Omron CX-Programmer project NewProject (CX-Programmer 9.73)

# PLC NewPLC1: CP1L M

## Global symbols (name address type ; comment)
100.03 BOOL  ; SOAP_APPLICATION
100.04 BOOL  ; BRUSHING
0.05 BOOL  ; SENSOR_5
0.00 BOOL  ; ON_START
0.01 BOOL  ; SENSOR_1
0.02 BOOL  ; SENSOR_2
0.03 BOOL  ; SENSOR_3
0.04 BOOL  ; SENSOR_4
0.06 BOOL  ; STOP_BUTTON
100.00 BOOL  ; INDIKATOR_LAMP
100.01 BOOL  ; KONVEYOR
100.02 BOOL  ; WATER_SPRAYER
100.05 BOOL  ; WATER_WASHER
100.06 BOOL  ; DRYER
T0001 BOOL  ; T1
T0002 BOOL  ; T2
T0003 BOOL  ; T3
T0004 BOOL  ; T4
W100.00 BOOL  ; 0
W100.01 BOOL  ; 1
W100.05 BOOL  ; STOP

## Program NewProgram1 (cyclic task 0)

### Section Section1

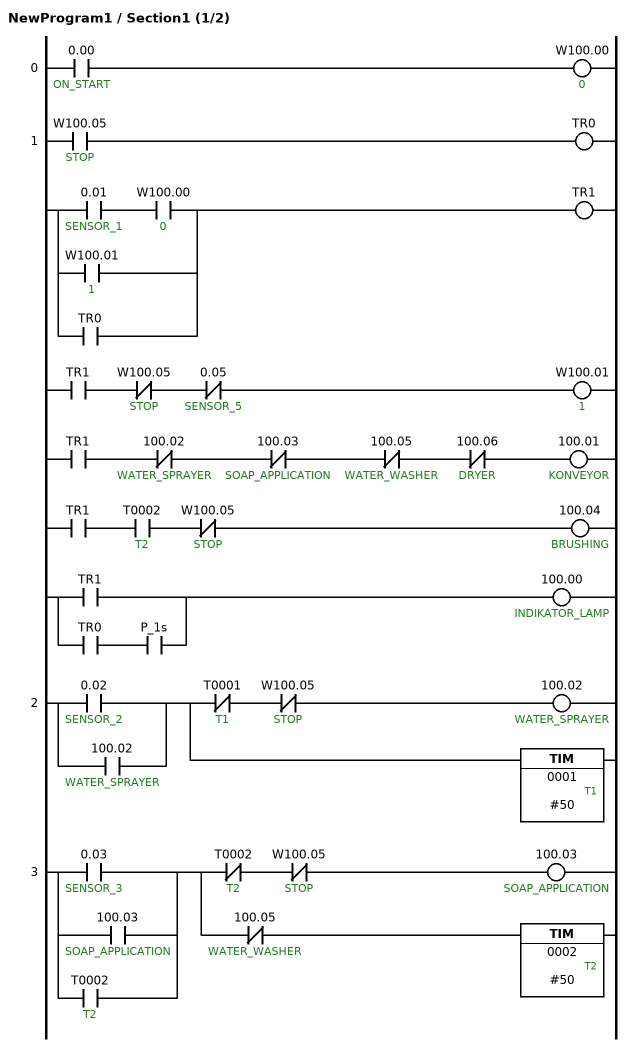
; rung 0
LD 0.00  ; ON_START
OUT W100.00  ; 0
; rung 1
LD 0.01  ; SENSOR_1
AND W100.00  ; 0
OR W100.01  ; 1
LD W100.05  ; STOP
OUT TR0
ORLD
OUT TR1
ANDNOT W100.05  ; STOP
ANDNOT 0.05  ; SENSOR_5
OUT W100.01  ; 1
LD TR1
ANDNOT 100.02  ; WATER_SPRAYER
ANDNOT 100.03  ; SOAP_APPLICATION
ANDNOT 100.05  ; WATER_WASHER
ANDNOT 100.06  ; DRYER
OUT 100.01  ; KONVEYOR
LD TR1
AND T0002  ; T2
ANDNOT W100.05  ; STOP
OUT 100.04  ; BRUSHING
LD TR1
LD TR0
AND P_1s
ORLD
OUT 100.00  ; INDIKATOR_LAMP
; rung 2
LD 0.02  ; SENSOR_2
OR 100.02  ; WATER_SPRAYER
OUT TR0
ANDNOT T0001  ; T1
ANDNOT W100.05  ; STOP
OUT 100.02  ; WATER_SPRAYER
LD TR0
TIM 0001 #50  ; T1
; rung 3
LD 0.03  ; SENSOR_3
OR 100.03  ; SOAP_APPLICATION
OR T0002  ; T2
OUT TR0
ANDNOT T0002  ; T2
ANDNOT W100.05  ; STOP
OUT 100.03  ; SOAP_APPLICATION
LD TR0
ANDNOT 100.05  ; WATER_WASHER
TIM 0002 #50  ; T2

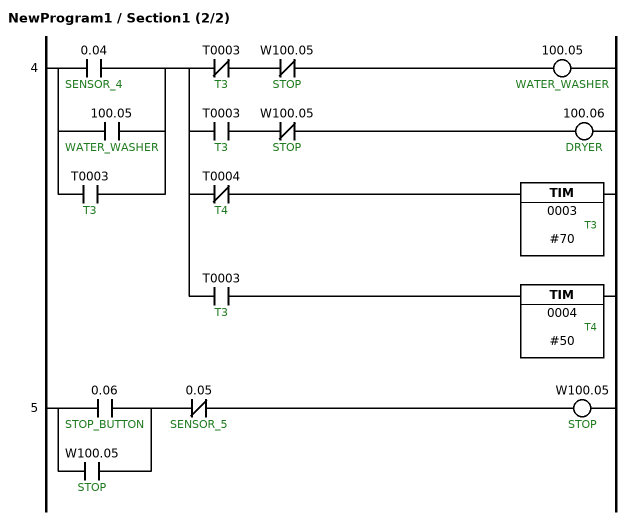
; rung 4
LD 0.04  ; SENSOR_4
OR 100.05  ; WATER_WASHER
OR T0003  ; T3
OUT TR0
ANDNOT T0003  ; T3
ANDNOT W100.05  ; STOP
OUT 100.05  ; WATER_WASHER
LD TR0
AND T0003  ; T3
ANDNOT W100.05  ; STOP
OUT 100.06  ; DRYER
LD TR0
ANDNOT T0004  ; T4
TIM 0003 #70  ; T3
LD TR0
AND T0003  ; T3
TIM 0004 #50  ; T4
; rung 5
LD 0.06  ; STOP_BUTTON
OR W100.05  ; STOP
ANDNOT 0.05  ; SENSOR_5
OUT W100.05  ; STOP

### Section END
; rung 0
END(001)